// TwinCAT 3 PLC project Motor_test
// ProgramVersion: 3.1.4024.0
// libraries:
//   Tc2_MC2, * (Beckhoff Automation GmbH)
//   Tc2_Standard, * (Beckhoff Automation GmbH)
//   Tc2_System, * (Beckhoff Automation GmbH)
//   Tc3_Module, * (Beckhoff Automation GmbH)
// project tree:
//   / PlcTask.TcTTO
//   POUs/ MAIN.TcPOU

CONFIGURATION Motor_test
    RESOURCE PLC ON TwinCAT3
        TASK PlcTask(INTERVAL := T#10ms, PRIORITY := 22);
        PROGRAM MAIN WITH PlcTask : MAIN;
    END_RESOURCE
END_CONFIGURATION

// ---- POUs/MAIN.TcPOU
PROGRAM MAIN
VAR
Xas: AXIS_REF;
Yas: AXIS_REF;

XMotorPower: MC_power; 
YMotorPower: MC_power;
XMotorPosition: MC_MoveAbsolute;
YMotorPosition: MC_MoveAbsolute;
XMotorHome: MC_Home;
YMotorHome: MC_Home;
Estop AT %I*: BOOL;
links: BOOL;
rechts: BOOL;
XMotorReset: MC_Reset;
YMotorReset: MC_Reset;

END_VAR

XMotorPosition(Axis := Xas, Velocity := 250, Acceleration := 10, Deceleration := 2000, Jerk := 100000);
YMotorPosition(Axis := Yas, Velocity := 250, Acceleration := 10, Deceleration := 2000, Jerk := 100000);
XMotorPower(Axis:= Xas, Enable := TRUE, Enable_Positive := TRUE, Enable_Negative := TRUE);
YMotorPower(Axis:= Yas, Enable := TRUE, Enable_Positive := TRUE, Enable_Negative := TRUE);


//XMotorHome(Axis := Xas, Execute := TRUE, Position := 0, HomingMode := MC_DIRECT); 

IF links AND NOT rechts AND Estop THEN
	XMotorPosition(Axis := Xas, Execute := TRUE, Position:= 500);
END_IF

IF NOT links AND rechts AND Estop THEN
	XMotorPosition(Axis := Xas, Execute := TRUE, Position:= -500);
END_IF

IF NOT Estop THEN
	XMotorPosition( Axis := Xas, Execute := FALSE);
END_IF

END_PROGRAM
